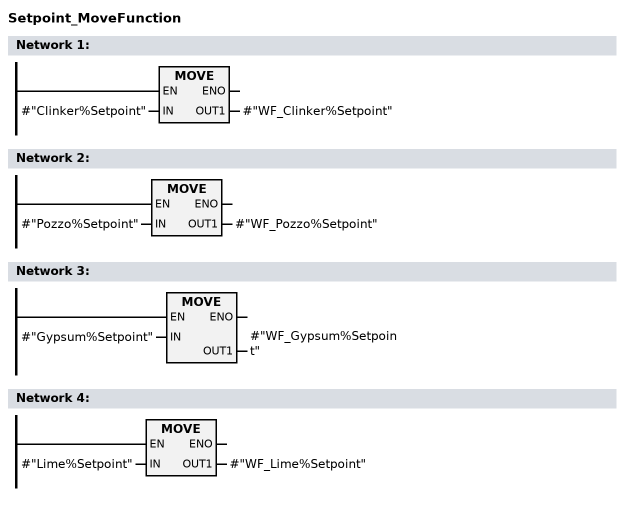
   RUNG wire#powerrail
      Move(in := #"Clinker%Setpoint", out1 => #"WF_Clinker%Setpoint")
   END_RUNG
   // the same network as SCL:
   #"WF_Clinker%Setpoint" := #"Clinker%Setpoint";
END_REGION

REGION Network 2
   RUNG wire#powerrail
      Move(in := #"Pozzo%Setpoint", out1 => #"WF_Pozzo%Setpoint")
   END_RUNG
   // the same network as SCL:
   #"WF_Pozzo%Setpoint" := #"Pozzo%Setpoint";
END_REGION

REGION Network 3
   RUNG wire#powerrail
      Move(in := #"Gypsum%Setpoint", out1 => #"WF_Gypsum%Setpoint")
   END_RUNG
   // the same network as SCL:
   #"WF_Gypsum%Setpoint" := #"Gypsum%Setpoint";
END_REGION

REGION Network 4
   RUNG wire#powerrail
      Move(in := #"Lime%Setpoint", out1 => #"WF_Lime%Setpoint")
   END_RUNG
   // the same network as SCL:
   #"WF_Lime%Setpoint" := #"Lime%Setpoint";
END_REGION
END_FUNCTION

FUNCTION "SelectionIndication" : Void   // FC10, LAD
{ S7_Optimized_Access := 'TRUE' }
VERSION : 0.1
   VAR_INPUT
      CementType_Selected : Bool;
      "Inretlock 1" : Bool;
      "Inretlock 2" : Bool;
      "Inretlock 3" : Bool;
   END_VAR
   VAR_IN_OUT
      Selected : Bool;
   END_VAR
BEGIN

REGION Network 1: Selecting Material Type
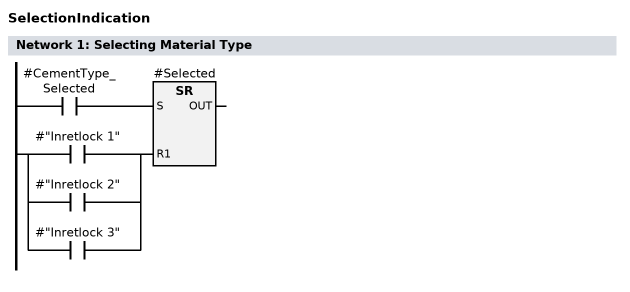
   RUNG wire#powerrail
      Contact( #CementType_Selected )
      S_SR(operand := #Selected, r1 := wire#w1)
   END_RUNG
   RUNG wire#powerrail
      Contact( #"Inretlock 1" )
   END_RUNG wire#w1
   RUNG wire#powerrail
      Contact( #"Inretlock 2" )
   END_RUNG wire#w1
   RUNG wire#powerrail
      Contact( #"Inretlock 3" )
   END_RUNG wire#w1
   // the same network as SCL:
   IF #CementType_Selected THEN
       #Selected := TRUE;   // SR flip-flop
   END_IF;
   IF #"Inretlock 1" OR #"Inretlock 2" OR #"Inretlock 3" THEN #Selected := FALSE; END_IF;
END_REGION
END_FUNCTION

ORGANIZATION_BLOCK "PIDFunctions"   // OB30, LAD, CyclicInterrupt
{ S7_Optimized_Access := 'TRUE' }
VERSION : 0.1
   VAR_INPUT
      Initial_Call : Bool;   // Initial call of this OB
      Event_Count : Int;   // Events discarded
   END_VAR
BEGIN

REGION Network 1: CLINKER BLOCK
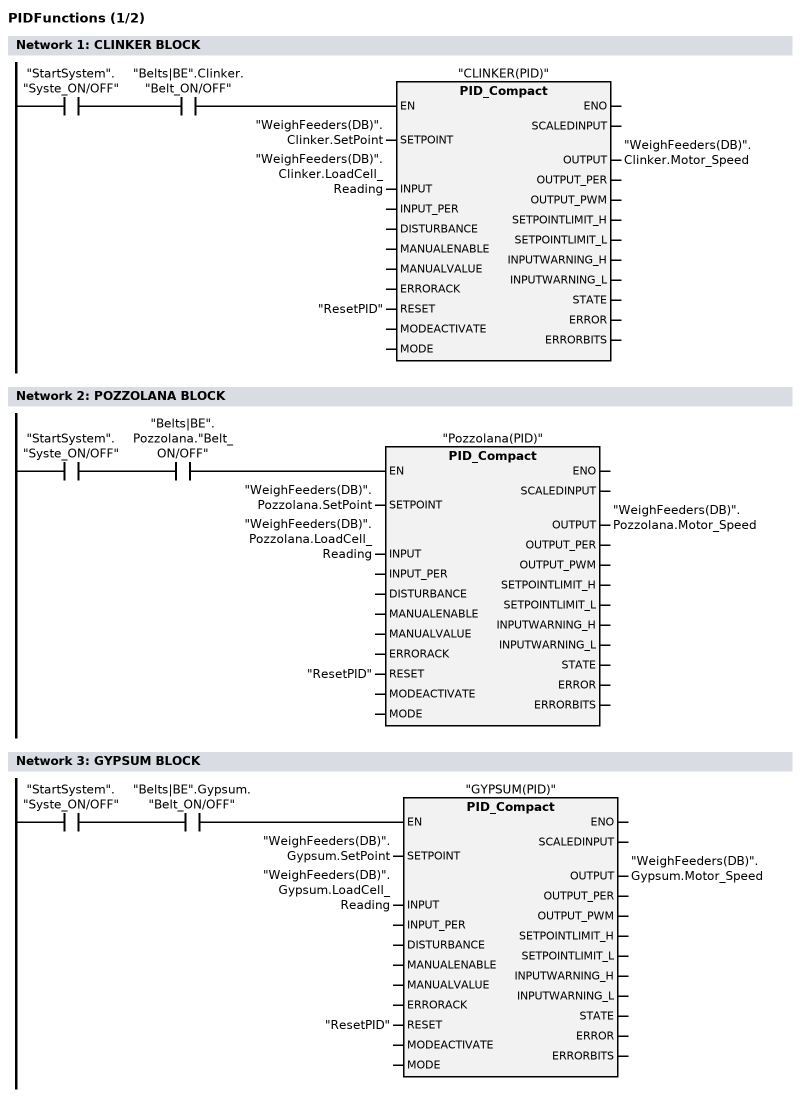
   IF "StartSystem"."Syste_ON/OFF" AND "Belts|BE".Clinker."Belt_ON/OFF" THEN
       "CLINKER(PID)"(Setpoint := "WeighFeeders(DB)".Clinker.SetPoint,   // PID_Compact
                      Input := "WeighFeeders(DB)".Clinker.LoadCell_Reading,
                      Reset := "ResetPID",
                      Output => "WeighFeeders(DB)".Clinker.Motor_Speed);
   END_IF;
END_REGION

REGION Network 2: POZZOLANA BLOCK
   IF "StartSystem"."Syste_ON/OFF" AND "Belts|BE".Pozzolana."Belt_ON/OFF" THEN
       "Pozzolana(PID)"(Setpoint := "WeighFeeders(DB)".Pozzolana.SetPoint,   // PID_Compact
                        Input := "WeighFeeders(DB)".Pozzolana.LoadCell_Reading,
                        Reset := "ResetPID",
                        Output => "WeighFeeders(DB)".Pozzolana.Motor_Speed);
   END_IF;
END_REGION

REGION Network 3: GYPSUM BLOCK
   IF "StartSystem"."Syste_ON/OFF" AND "Belts|BE".Gypsum."Belt_ON/OFF" THEN
       "GYPSUM(PID)"(Setpoint := "WeighFeeders(DB)".Gypsum.SetPoint,   // PID_Compact
                     Input := "WeighFeeders(DB)".Gypsum.LoadCell_Reading,
                     Reset := "ResetPID",
                     Output => "WeighFeeders(DB)".Gypsum.Motor_Speed);
   END_IF;
END_REGION

REGION Network 4: LIMESTONE BLOCK
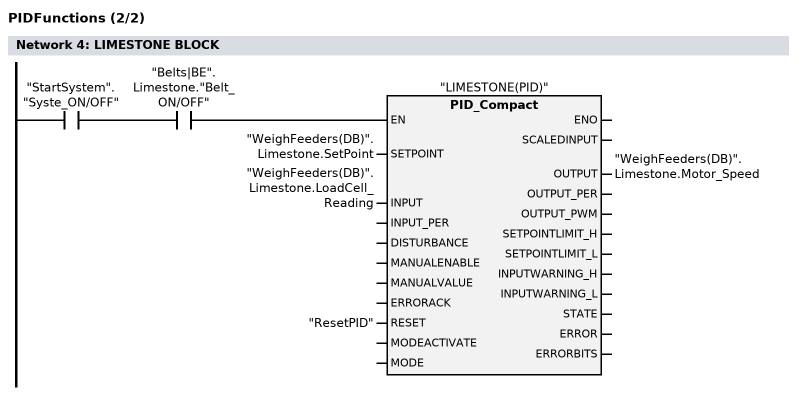
   IF "StartSystem"."Syste_ON/OFF" AND "Belts|BE".Limestone."Belt_ON/OFF" THEN
       "LIMESTONE(PID)"(Setpoint := "WeighFeeders(DB)".Limestone.SetPoint,   // PID_Compact
                        Input := "WeighFeeders(DB)".Limestone.LoadCell_Reading,
                        Reset := "ResetPID",
                        Output => "WeighFeeders(DB)".Limestone.Motor_Speed);
   END_IF;
END_REGION
END_ORGANIZATION_BLOCK

ORGANIZATION_BLOCK "LoadCell_Simulation(0.1s)"   // OB31, LAD, CyclicInterrupt
{ S7_Optimized_Access := 'TRUE' }
VERSION : 0.1
   VAR_INPUT
      Initial_Call : Bool;   // Initial call of this OB
      Event_Count : Int;   // Events discarded
   END_VAR
BEGIN

REGION Network 1: CLINKER
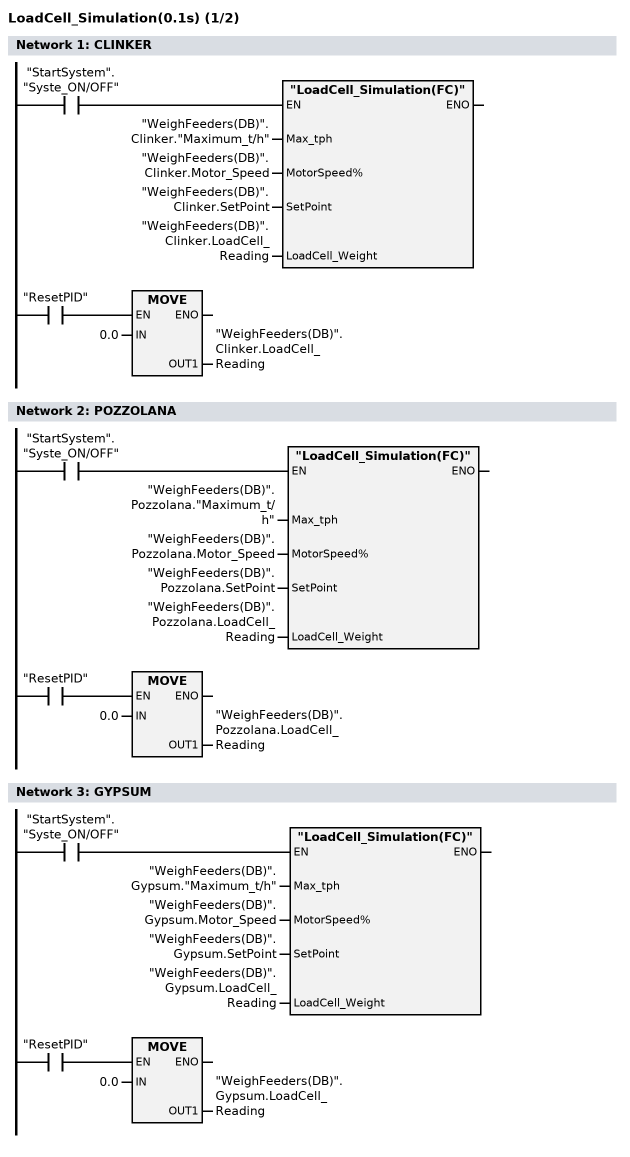
   RUNG wire#powerrail
      Contact( "StartSystem"."Syste_ON/OFF" )
      "LoadCell_Simulation(FC)"(Max_tph := "WeighFeeders(DB)".Clinker."Maximum_t/h", "MotorSpeed%" := "WeighFeeders(DB)".Clinker.Motor_Speed, SetPoint := "WeighFeeders(DB)".Clinker.SetPoint, LoadCell_Weight := "WeighFeeders(DB)".Clinker.LoadCell_Reading)
   END_RUNG
   RUNG wire#powerrail
      Contact( "ResetPID" )
      Move(in := 0.0, out1 => "WeighFeeders(DB)".Clinker.LoadCell_Reading)
   END_RUNG
   // the same network as SCL:
   IF "StartSystem"."Syste_ON/OFF" THEN
       "LoadCell_Simulation(FC)"(Max_tph := "WeighFeeders(DB)".Clinker."Maximum_t/h",
                               "MotorSpeed%" := "WeighFeeders(DB)".Clinker.Motor_Speed,
                               SetPoint := "WeighFeeders(DB)".Clinker.SetPoint,
                               LoadCell_Weight := "WeighFeeders(DB)".Clinker.LoadCell_Reading);
   END_IF;
   IF "ResetPID" THEN "WeighFeeders(DB)".Clinker.LoadCell_Reading := 0.0; END_IF;
END_REGION

REGION Network 2: POZZOLANA
   RUNG wire#powerrail
      Contact( "StartSystem"."Syste_ON/OFF" )
      "LoadCell_Simulation(FC)"(Max_tph := "WeighFeeders(DB)".Pozzolana."Maximum_t/h", "MotorSpeed%" := "WeighFeeders(DB)".Pozzolana.Motor_Speed, SetPoint := "WeighFeeders(DB)".Pozzolana.SetPoint, LoadCell_Weight := "WeighFeeders(DB)".Pozzolana.LoadCell_Reading)
   END_RUNG
   RUNG wire#powerrail
      Contact( "ResetPID" )
      Move(in := 0.0, out1 => "WeighFeeders(DB)".Pozzolana.LoadCell_Reading)
   END_RUNG
   // the same network as SCL:
   IF "StartSystem"."Syste_ON/OFF" THEN
       "LoadCell_Simulation(FC)"(Max_tph := "WeighFeeders(DB)".Pozzolana."Maximum_t/h",
                               "MotorSpeed%" := "WeighFeeders(DB)".Pozzolana.Motor_Speed,
                               SetPoint := "WeighFeeders(DB)".Pozzolana.SetPoint,
                               LoadCell_Weight := "WeighFeeders(DB)".Pozzolana.LoadCell_Reading);
   END_IF;
   IF "ResetPID" THEN "WeighFeeders(DB)".Pozzolana.LoadCell_Reading := 0.0; END_IF;
END_REGION

REGION Network 3: GYPSUM
   RUNG wire#powerrail
      Contact( "StartSystem"."Syste_ON/OFF" )
      "LoadCell_Simulation(FC)"(Max_tph := "WeighFeeders(DB)".Gypsum."Maximum_t/h", "MotorSpeed%" := "WeighFeeders(DB)".Gypsum.Motor_Speed, SetPoint := "WeighFeeders(DB)".Gypsum.SetPoint, LoadCell_Weight := "WeighFeeders(DB)".Gypsum.LoadCell_Reading)
   END_RUNG
   RUNG wire#powerrail
      Contact( "ResetPID" )
      Move(in := 0.0, out1 => "WeighFeeders(DB)".Gypsum.LoadCell_Reading)
   END_RUNG
   // the same network as SCL:
   IF "StartSystem"."Syste_ON/OFF" THEN
       "LoadCell_Simulation(FC)"(Max_tph := "WeighFeeders(DB)".Gypsum."Maximum_t/h",
                               "MotorSpeed%" := "WeighFeeders(DB)".Gypsum.Motor_Speed,
                               SetPoint := "WeighFeeders(DB)".Gypsum.SetPoint,
                               LoadCell_Weight := "WeighFeeders(DB)".Gypsum.LoadCell_Reading);
   END_IF;
   IF "ResetPID" THEN "WeighFeeders(DB)".Gypsum.LoadCell_Reading := 0.0; END_IF;
END_REGION

REGION Network 4: LIMESTONE
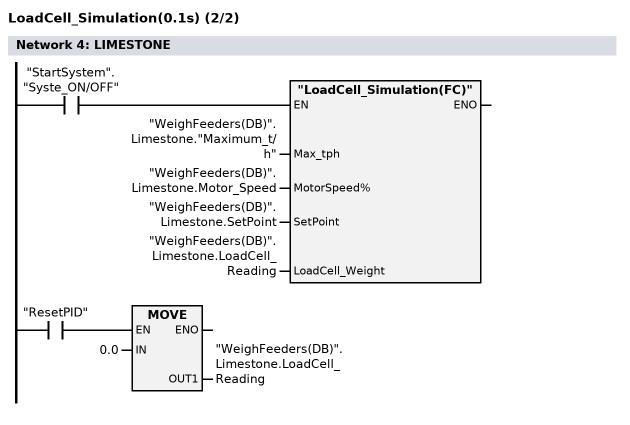
   RUNG wire#powerrail
      Contact( "StartSystem"."Syste_ON/OFF" )
      "LoadCell_Simulation(FC)"(Max_tph := "WeighFeeders(DB)".Limestone."Maximum_t/h", "MotorSpeed%" := "WeighFeeders(DB)".Limestone.Motor_Speed, SetPoint := "WeighFeeders(DB)".Limestone.SetPoint, LoadCell_Weight := "WeighFeeders(DB)".Limestone.LoadCell_Reading)
   END_RUNG
   RUNG wire#powerrail
      Contact( "ResetPID" )
      Move(in := 0.0, out1 => "WeighFeeders(DB)".Limestone.LoadCell_Reading)
   END_RUNG
   // the same network as SCL:
   IF "StartSystem"."Syste_ON/OFF" THEN
       "LoadCell_Simulation(FC)"(Max_tph := "WeighFeeders(DB)".Limestone."Maximum_t/h",
                               "MotorSpeed%" := "WeighFeeders(DB)".Limestone.Motor_Speed,
                               SetPoint := "WeighFeeders(DB)".Limestone.SetPoint,
                               LoadCell_Weight := "WeighFeeders(DB)".Limestone.LoadCell_Reading);
   END_IF;
   IF "ResetPID" THEN "WeighFeeders(DB)".Limestone.LoadCell_Reading := 0.0; END_IF;
END_REGION
END_ORGANIZATION_BLOCK

ORGANIZATION_BLOCK "Cement_TypesSelection"   // OB33, LAD, CyclicInterrupt
{ S7_Optimized_Access := 'TRUE' }
VERSION : 0.1
   VAR_INPUT
      Initial_Call : Bool;   // Initial call of this OB
      Event_Count : Int;   // Events discarded
   END_VAR
BEGIN

REGION Network 1: KP_Silver Selection Indicator
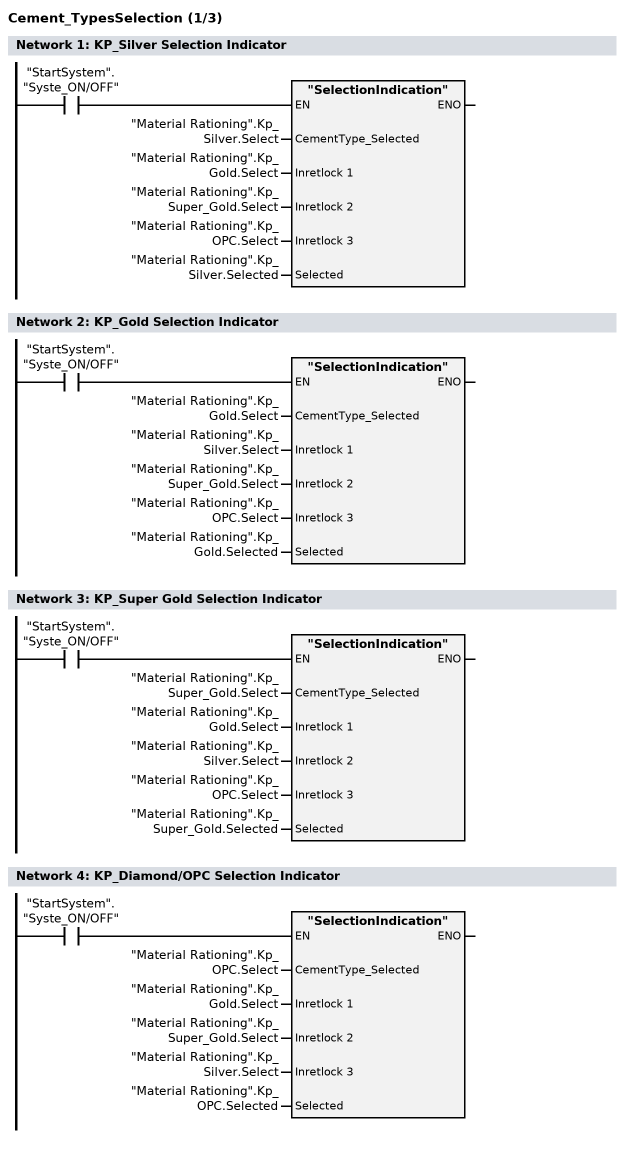
   RUNG wire#powerrail
      Contact( "StartSystem"."Syste_ON/OFF" )
      "SelectionIndication"(CementType_Selected := "Material Rationing".Kp_Silver.Select, "Inretlock 1" := "Material Rationing".Kp_Gold.Select, "Inretlock 2" := "Material Rationing".Kp_Super_Gold.Select, "Inretlock 3" := "Material Rationing".Kp_OPC.Select, Selected := "Material Rationing".Kp_Silver.Selected)
   END_RUNG
   // the same network as SCL:
   IF "StartSystem"."Syste_ON/OFF" THEN
       "SelectionIndication"(CementType_Selected := "Material Rationing".Kp_Silver.Select,
                             "Inretlock 1" := "Material Rationing".Kp_Gold.Select,
                             "Inretlock 2" := "Material Rationing".Kp_Super_Gold.Select,
                             "Inretlock 3" := "Material Rationing".Kp_OPC.Select,
                             Selected := "Material Rationing".Kp_Silver.Selected);
   END_IF;
END_REGION

REGION Network 2: KP_Gold Selection Indicator
   RUNG wire#powerrail
      Contact( "StartSystem"."Syste_ON/OFF" )
      "SelectionIndication"(CementType_Selected := "Material Rationing".Kp_Gold.Select, "Inretlock 1" := "Material Rationing".Kp_Silver.Select, "Inretlock 2" := "Material Rationing".Kp_Super_Gold.Select, "Inretlock 3" := "Material Rationing".Kp_OPC.Select, Selected := "Material Rationing".Kp_Gold.Selected)
   END_RUNG
   // the same network as SCL:
   IF "StartSystem"."Syste_ON/OFF" THEN
       "SelectionIndication"(CementType_Selected := "Material Rationing".Kp_Gold.Select,
                             "Inretlock 1" := "Material Rationing".Kp_Silver.Select,
                             "Inretlock 2" := "Material Rationing".Kp_Super_Gold.Select,
                             "Inretlock 3" := "Material Rationing".Kp_OPC.Select,
                             Selected := "Material Rationing".Kp_Gold.Selected);
   END_IF;
END_REGION

REGION Network 3: KP_Super Gold Selection Indicator
   RUNG wire#powerrail
      Contact( "StartSystem"."Syste_ON/OFF" )
      "SelectionIndication"(CementType_Selected := "Material Rationing".Kp_Super_Gold.Select, "Inretlock 1" := "Material Rationing".Kp_Gold.Select, "Inretlock 2" := "Material Rationing".Kp_Silver.Select, "Inretlock 3" := "Material Rationing".Kp_OPC.Select, Selected := "Material Rationing".Kp_Super_Gold.Selected)
   END_RUNG
   // the same network as SCL:
   IF "StartSystem"."Syste_ON/OFF" THEN
       "SelectionIndication"(CementType_Selected := "Material Rationing".Kp_Super_Gold.Select,
                             "Inretlock 1" := "Material Rationing".Kp_Gold.Select,
                             "Inretlock 2" := "Material Rationing".Kp_Silver.Select,
                             "Inretlock 3" := "Material Rationing".Kp_OPC.Select,
                             Selected := "Material Rationing".Kp_Super_Gold.Selected);
   END_IF;
END_REGION

REGION Network 4: KP_Diamond/OPC Selection Indicator
   RUNG wire#powerrail
      Contact( "StartSystem"."Syste_ON/OFF" )
      "SelectionIndication"(CementType_Selected := "Material Rationing".Kp_OPC.Select, "Inretlock 1" := "Material Rationing".Kp_Gold.Select, "Inretlock 2" := "Material Rationing".Kp_Super_Gold.Select, "Inretlock 3" := "Material Rationing".Kp_Silver.Select, Selected := "Material Rationing".Kp_OPC.Selected)
   END_RUNG
   // the same network as SCL:
   IF "StartSystem"."Syste_ON/OFF" THEN
       "SelectionIndication"(CementType_Selected := "Material Rationing".Kp_OPC.Select,
                             "Inretlock 1" := "Material Rationing".Kp_Gold.Select,
                             "Inretlock 2" := "Material Rationing".Kp_Super_Gold.Select,
                             "Inretlock 3" := "Material Rationing".Kp_Silver.Select,
                             Selected := "Material Rationing".Kp_OPC.Selected);
   END_IF;
END_REGION

REGION Network 5: If Kp_Silver has been selected the setpoint is calculated in this block
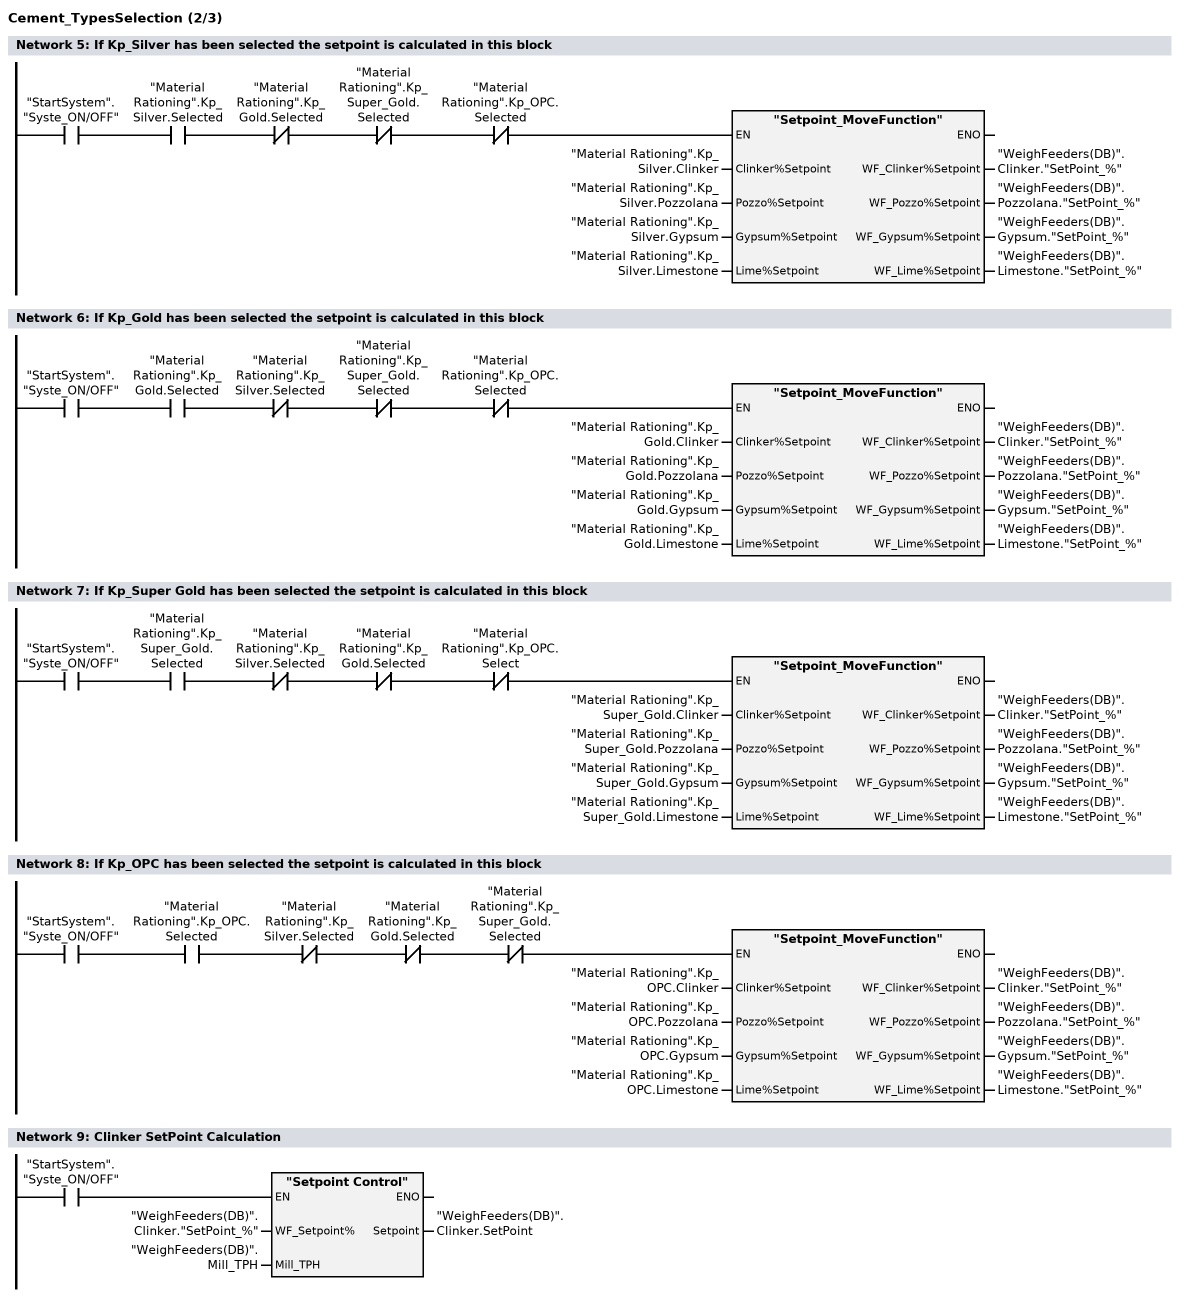
   RUNG wire#powerrail
      Contact( "StartSystem"."Syste_ON/OFF" )
      Contact( "Material Rationing".Kp_Silver.Selected )
      I_Contact( "Material Rationing".Kp_Gold.Selected )
      I_Contact( "Material Rationing".Kp_Super_Gold.Selected )
      I_Contact( "Material Rationing".Kp_OPC.Selected )
      "Setpoint_MoveFunction"("Clinker%Setpoint" := "Material Rationing".Kp_Silver.Clinker, "Pozzo%Setpoint" := "Material Rationing".Kp_Silver.Pozzolana, "Gypsum%Setpoint" := "Material Rationing".Kp_Silver.Gypsum, "Lime%Setpoint" := "Material Rationing".Kp_Silver.Limestone, "WF_Clinker%Setpoint" => "WeighFeeders(DB)".Clinker."SetPoint_%", "WF_Pozzo%Setpoint" => "WeighFeeders(DB)".Pozzolana."SetPoint_%", "WF_Gypsum%Setpoint" => "WeighFeeders(DB)".Gypsum."SetPoint_%", "WF_Lime%Setpoint" => "WeighFeeders(DB)".Limestone."SetPoint_%")
   END_RUNG
   // the same network as SCL:
   IF "StartSystem"."Syste_ON/OFF" AND "Material Rationing".Kp_Silver.Selected AND NOT "Material Rationing".Kp_Gold.Selected AND NOT "Material Rationing".Kp_Super_Gold.Selected AND NOT "Material Rationing".Kp_OPC.Selected THEN
       "Setpoint_MoveFunction"("Clinker%Setpoint" := "Material Rationing".Kp_Silver.Clinker,
                               "Pozzo%Setpoint" := "Material Rationing".Kp_Silver.Pozzolana,
                               "Gypsum%Setpoint" := "Material Rationing".Kp_Silver.Gypsum,
                               "Lime%Setpoint" := "Material Rationing".Kp_Silver.Limestone,
                               "WF_Clinker%Setpoint" => "WeighFeeders(DB)".Clinker."SetPoint_%",
                               "WF_Pozzo%Setpoint" => "WeighFeeders(DB)".Pozzolana."SetPoint_%",
                               "WF_Gypsum%Setpoint" => "WeighFeeders(DB)".Gypsum."SetPoint_%",
                               "WF_Lime%Setpoint" => "WeighFeeders(DB)".Limestone."SetPoint_%");
   END_IF;
END_REGION

REGION Network 6: If Kp_Gold has been selected the setpoint is calculated in this block
   RUNG wire#powerrail
      Contact( "StartSystem"."Syste_ON/OFF" )
      Contact( "Material Rationing".Kp_Gold.Selected )
      I_Contact( "Material Rationing".Kp_Silver.Selected )
      I_Contact( "Material Rationing".Kp_Super_Gold.Selected )
      I_Contact( "Material Rationing".Kp_OPC.Selected )
      "Setpoint_MoveFunction"("Clinker%Setpoint" := "Material Rationing".Kp_Gold.Clinker, "Pozzo%Setpoint" := "Material Rationing".Kp_Gold.Pozzolana, "Gypsum%Setpoint" := "Material Rationing".Kp_Gold.Gypsum, "Lime%Setpoint" := "Material Rationing".Kp_Gold.Limestone, "WF_Clinker%Setpoint" => "WeighFeeders(DB)".Clinker."SetPoint_%", "WF_Pozzo%Setpoint" => "WeighFeeders(DB)".Pozzolana."SetPoint_%", "WF_Gypsum%Setpoint" => "WeighFeeders(DB)".Gypsum."SetPoint_%", "WF_Lime%Setpoint" => "WeighFeeders(DB)".Limestone."SetPoint_%")
   END_RUNG
   // the same network as SCL:
   IF "StartSystem"."Syste_ON/OFF" AND "Material Rationing".Kp_Gold.Selected AND NOT "Material Rationing".Kp_Silver.Selected AND NOT "Material Rationing".Kp_Super_Gold.Selected AND NOT "Material Rationing".Kp_OPC.Selected THEN
       "Setpoint_MoveFunction"("Clinker%Setpoint" := "Material Rationing".Kp_Gold.Clinker,
                               "Pozzo%Setpoint" := "Material Rationing".Kp_Gold.Pozzolana,
                               "Gypsum%Setpoint" := "Material Rationing".Kp_Gold.Gypsum,
                               "Lime%Setpoint" := "Material Rationing".Kp_Gold.Limestone,
                               "WF_Clinker%Setpoint" => "WeighFeeders(DB)".Clinker."SetPoint_%",
                               "WF_Pozzo%Setpoint" => "WeighFeeders(DB)".Pozzolana."SetPoint_%",
                               "WF_Gypsum%Setpoint" => "WeighFeeders(DB)".Gypsum."SetPoint_%",
                               "WF_Lime%Setpoint" => "WeighFeeders(DB)".Limestone."SetPoint_%");
   END_IF;
END_REGION

REGION Network 7: If Kp_Super Gold has been selected the setpoint is calculated in this block
   RUNG wire#powerrail
      Contact( "StartSystem"."Syste_ON/OFF" )
      Contact( "Material Rationing".Kp_Super_Gold.Selected )
      I_Contact( "Material Rationing".Kp_Silver.Selected )
      I_Contact( "Material Rationing".Kp_Gold.Selected )
      I_Contact( "Material Rationing".Kp_OPC.Select )
      "Setpoint_MoveFunction"("Clinker%Setpoint" := "Material Rationing".Kp_Super_Gold.Clinker, "Pozzo%Setpoint" := "Material Rationing".Kp_Super_Gold.Pozzolana, "Gypsum%Setpoint" := "Material Rationing".Kp_Super_Gold.Gypsum, "Lime%Setpoint" := "Material Rationing".Kp_Super_Gold.Limestone, "WF_Clinker%Setpoint" => "WeighFeeders(DB)".Clinker."SetPoint_%", "WF_Pozzo%Setpoint" => "WeighFeeders(DB)".Pozzolana."SetPoint_%", "WF_Gypsum%Setpoint" => "WeighFeeders(DB)".Gypsum."SetPoint_%", "WF_Lime%Setpoint" => "WeighFeeders(DB)".Limestone."SetPoint_%")
   END_RUNG
   // the same network as SCL:
   IF "StartSystem"."Syste_ON/OFF" AND "Material Rationing".Kp_Super_Gold.Selected AND NOT "Material Rationing".Kp_Silver.Selected AND NOT "Material Rationing".Kp_Gold.Selected AND NOT "Material Rationing".Kp_OPC.Select THEN
       "Setpoint_MoveFunction"("Clinker%Setpoint" := "Material Rationing".Kp_Super_Gold.Clinker,
                               "Pozzo%Setpoint" := "Material Rationing".Kp_Super_Gold.Pozzolana,
                               "Gypsum%Setpoint" := "Material Rationing".Kp_Super_Gold.Gypsum,
                               "Lime%Setpoint" := "Material Rationing".Kp_Super_Gold.Limestone,
                               "WF_Clinker%Setpoint" => "WeighFeeders(DB)".Clinker."SetPoint_%",
                               "WF_Pozzo%Setpoint" => "WeighFeeders(DB)".Pozzolana."SetPoint_%",
                               "WF_Gypsum%Setpoint" => "WeighFeeders(DB)".Gypsum."SetPoint_%",
                               "WF_Lime%Setpoint" => "WeighFeeders(DB)".Limestone."SetPoint_%");
   END_IF;
END_REGION

REGION Network 8: If Kp_OPC has been selected the setpoint is calculated in this block
   RUNG wire#powerrail
      Contact( "StartSystem"."Syste_ON/OFF" )
      Contact( "Material Rationing".Kp_OPC.Selected )
      I_Contact( "Material Rationing".Kp_Silver.Selected )
      I_Contact( "Material Rationing".Kp_Gold.Selected )
      I_Contact( "Material Rationing".Kp_Super_Gold.Selected )
      "Setpoint_MoveFunction"("Clinker%Setpoint" := "Material Rationing".Kp_OPC.Clinker, "Pozzo%Setpoint" := "Material Rationing".Kp_OPC.Pozzolana, "Gypsum%Setpoint" := "Material Rationing".Kp_OPC.Gypsum, "Lime%Setpoint" := "Material Rationing".Kp_OPC.Limestone, "WF_Clinker%Setpoint" => "WeighFeeders(DB)".Clinker."SetPoint_%", "WF_Pozzo%Setpoint" => "WeighFeeders(DB)".Pozzolana."SetPoint_%", "WF_Gypsum%Setpoint" => "WeighFeeders(DB)".Gypsum."SetPoint_%", "WF_Lime%Setpoint" => "WeighFeeders(DB)".Limestone."SetPoint_%")
   END_RUNG
   // the same network as SCL:
   IF "StartSystem"."Syste_ON/OFF" AND "Material Rationing".Kp_OPC.Selected AND NOT "Material Rationing".Kp_Silver.Selected AND NOT "Material Rationing".Kp_Gold.Selected AND NOT "Material Rationing".Kp_Super_Gold.Selected THEN
       "Setpoint_MoveFunction"("Clinker%Setpoint" := "Material Rationing".Kp_OPC.Clinker,
                               "Pozzo%Setpoint" := "Material Rationing".Kp_OPC.Pozzolana,
                               "Gypsum%Setpoint" := "Material Rationing".Kp_OPC.Gypsum,
                               "Lime%Setpoint" := "Material Rationing".Kp_OPC.Limestone,
                               "WF_Clinker%Setpoint" => "WeighFeeders(DB)".Clinker."SetPoint_%",
                               "WF_Pozzo%Setpoint" => "WeighFeeders(DB)".Pozzolana."SetPoint_%",
                               "WF_Gypsum%Setpoint" => "WeighFeeders(DB)".Gypsum."SetPoint_%",
                               "WF_Lime%Setpoint" => "WeighFeeders(DB)".Limestone."SetPoint_%");
   END_IF;
END_REGION

REGION Network 9: Clinker SetPoint Calculation
   RUNG wire#powerrail
      Contact( "StartSystem"."Syste_ON/OFF" )
      "Setpoint Control"("WF_Setpoint%" := "WeighFeeders(DB)".Clinker."SetPoint_%", Mill_TPH := "WeighFeeders(DB)".Mill_TPH, Setpoint => "WeighFeeders(DB)".Clinker.SetPoint)
   END_RUNG
   // the same network as SCL:
   IF "StartSystem"."Syste_ON/OFF" THEN
       "Setpoint Control"("WF_Setpoint%" := "WeighFeeders(DB)".Clinker."SetPoint_%",
                          Mill_TPH := "WeighFeeders(DB)".Mill_TPH,
                          Setpoint => "WeighFeeders(DB)".Clinker.SetPoint);
   END_IF;
END_REGION

REGION Network 10: Pozzolana SetPoint Calculation
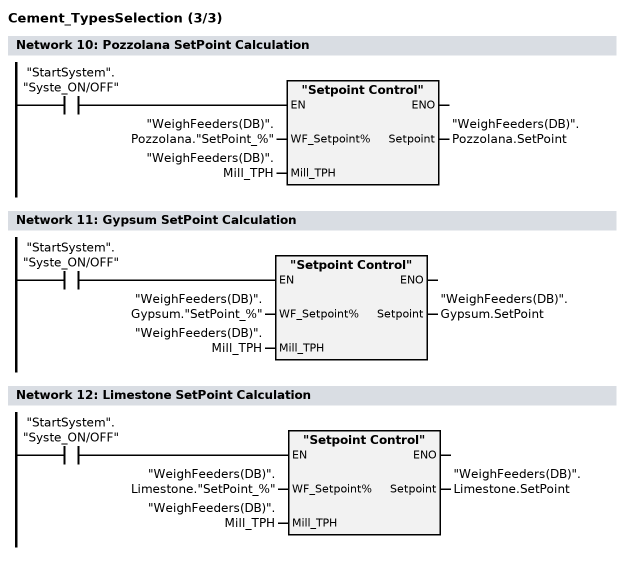
   RUNG wire#powerrail
      Contact( "StartSystem"."Syste_ON/OFF" )
      "Setpoint Control"("WF_Setpoint%" := "WeighFeeders(DB)".Pozzolana."SetPoint_%", Mill_TPH := "WeighFeeders(DB)".Mill_TPH, Setpoint => "WeighFeeders(DB)".Pozzolana.SetPoint)
   END_RUNG
   // the same network as SCL:
   IF "StartSystem"."Syste_ON/OFF" THEN
       "Setpoint Control"("WF_Setpoint%" := "WeighFeeders(DB)".Pozzolana."SetPoint_%",
                          Mill_TPH := "WeighFeeders(DB)".Mill_TPH,
                          Setpoint => "WeighFeeders(DB)".Pozzolana.SetPoint);
   END_IF;
END_REGION

REGION Network 11: Gypsum SetPoint Calculation
   RUNG wire#powerrail
      Contact( "StartSystem"."Syste_ON/OFF" )
      "Setpoint Control"("WF_Setpoint%" := "WeighFeeders(DB)".Gypsum."SetPoint_%", Mill_TPH := "WeighFeeders(DB)".Mill_TPH, Setpoint => "WeighFeeders(DB)".Gypsum.SetPoint)
   END_RUNG
   // the same network as SCL:
   IF "StartSystem"."Syste_ON/OFF" THEN
       "Setpoint Control"("WF_Setpoint%" := "WeighFeeders(DB)".Gypsum."SetPoint_%",
                          Mill_TPH := "WeighFeeders(DB)".Mill_TPH,
                          Setpoint => "WeighFeeders(DB)".Gypsum.SetPoint);
   END_IF;
END_REGION

REGION Network 12: Limestone SetPoint Calculation
   RUNG wire#powerrail
      Contact( "StartSystem"."Syste_ON/OFF" )
      "Setpoint Control"("WF_Setpoint%" := "WeighFeeders(DB)".Limestone."SetPoint_%", Mill_TPH := "WeighFeeders(DB)".Mill_TPH, Setpoint => "WeighFeeders(DB)".Limestone.SetPoint)
   END_RUNG
   // the same network as SCL:
   IF "StartSystem"."Syste_ON/OFF" THEN
       "Setpoint Control"("WF_Setpoint%" := "WeighFeeders(DB)".Limestone."SetPoint_%",
                          Mill_TPH := "WeighFeeders(DB)".Mill_TPH,
                          Setpoint => "WeighFeeders(DB)".Limestone.SetPoint);
   END_IF;
END_REGION
END_ORGANIZATION_BLOCK